// TIA Portal V17 export
// export: Created 2024-09-27T18:53:47.2459608Z, ExportSetting WithDefaults, DisplayName Totally Integrated Automation Portal, DisplayVersion V17, DisplayName TIA Portal Openness, DisplayVersion V17, DisplayName TIA Portal Version Control Interface, DisplayVersion V17, DisplayName STEP 7 Professional, DisplayVersion V17, DisplayName STEP 7 Safety, DisplayVersion V17, DisplayName WinCC Professional, DisplayVersion V17
FUNCTION "INFO" : Void   // FC7, LAD
{ S7_Optimized_Access := 'TRUE' }
VERSION : 0.1
// stored: AutoNumber true, IsIECCheckEnabled false, SetENOAutomatically false, UDAEnableTagReadback false
   VAR_TEMP
      temp_1 : Bool;
      m_temp2 : Bool;
      m_temp3 : Bool;
      m_temp4 : Bool;
      m_puls_liczniki : Bool;
      test1 : Bool;
   END_VAR
   VAR_TEMP   // added for the SCL form of the ladder/FBD networks
      _w1 : Bool;
   END_VAR
BEGIN

REGION Network 1: Powiadomienie o wykonaniu zadanej ilości sztuk
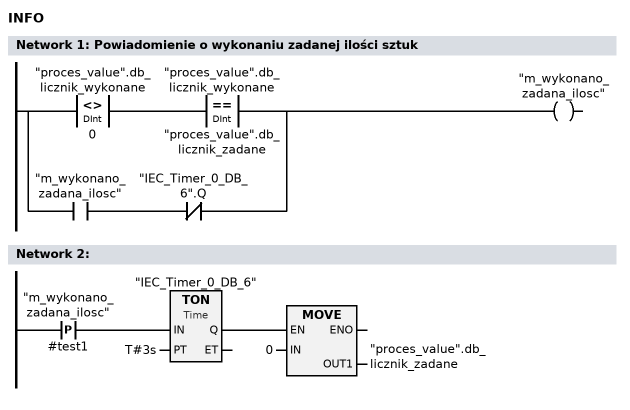
   RUNG wire#powerrail
      { S7_Templates := "SrcType := DInt" } NE_Contact(in1 := "proces_value".db_licznik_wykonane, in2 := 0)
      { S7_Templates := "SrcType := DInt" } EQ_Contact(in1 := "proces_value".db_licznik_wykonane, in2 := "proces_value".db_licznik_zadane)
      wire#w1
      Coil( "m_wykonano_zadana_ilosc" )
   END_RUNG
   RUNG wire#powerrail
      Contact( "m_wykonano_zadana_ilosc" )
      I_Contact( "IEC_Timer_0_DB_6".Q )
   END_RUNG wire#w1
   // the same network as SCL:
   "m_wykonano_zadana_ilosc" := (("proces_value".db_licznik_wykonane <> 0) AND ("proces_value".db_licznik_wykonane = "proces_value".db_licznik_zadane)) OR ("m_wykonano_zadana_ilosc" AND NOT "IEC_Timer_0_DB_6".Q);
END_REGION

REGION Network 2
   RUNG wire#powerrail
      P_Contact(operand := "m_wykonano_zadana_ilosc", bit := #test1)
      { S7_Templates := "time_type := Time" } "IEC_Timer_0_DB_6".TON(pt := T#3s, et =>)
      Move(in := 0, out1 => "proces_value".db_licznik_zadane)
   END_RUNG
   // the same network as SCL:
   #_w1 := "m_wykonano_zadana_ilosc" AND NOT #test1;   // rising edge of "m_wykonano_zadana_ilosc"
   #test1 := "m_wykonano_zadana_ilosc";
   "IEC_Timer_0_DB_6".TON(IN := #_w1, PT := T#3s);
   IF "IEC_Timer_0_DB_6".Q THEN "proces_value".db_licznik_zadane := 0; END_IF;
END_REGION

REGION Network 3: Info o Pauzie
END_REGION
END_FUNCTION
